{attribute 'GeneratedUsingTerminal: EL5101-0000-1020'}
{attribute addProperty BoxType "EL5101-0000-1020"}
{attribute addProperty Description "EL5101 1Ch. Inc. Encoder 5V"}
{attribute addProperty Physics "KK"}
{attribute addProperty Id "ENC_Status_compactAT %I*ENC_Status_compact_6F42455820ENC_Control_compactAT %Q*ENC_Control_compact_21E2D14D6WcStateAT %I*WcState_9091E0EB2InfoDataAT %I*InfoData_32EB74EA10"}
{attribute addProperty CRC "1729924372"}
{attribute addProperty Size "38"}
TYPE EL5101_671C8D14 EXTENDS EtcSlaveTerminalBase_947E5A46 :
STRUCT
	{attribute addProperty Name "ENC_Status_compact"}
	ENC_Status_compact : ENC_Status_compact_6F424558;
	{attribute addProperty Name "ENC_Control_compact"}
	ENC_Control_compact : ENC_Control_compact_21E2D14D;
	{attribute addProperty Name "WcState"}
	WcState : WcState_9091E0EB;
	{attribute addProperty Name "InfoData"}
	InfoData : InfoData_32EB74EA;
END_STRUCT
END_TYPE

(* stored: Version 1.2.0.0, ProductVersion 3.1.4024.11
   DUT EL5101_671C8D14: Id {52b80ddc-2c2d-49a7-aaf7-37d2555bdfa0} *)
